(* PLC project Generated.project, CODESYS CODESYS V3.5 SP19 Patch 1 *)
(* stored: creationDateTime 2026-09-06T13:00:42.426166, modificationDateTime 2026-09-06T13:00:42.426166 *)

(* values of E_Mode: DISABLE: Mode Désactivé / Veille de sécurité (sorties bloquées); MAINT_N1: Manuel Niveau 1 : Pilotage unitaire avec toutes sécurités actives; MAINT_N2: Manuel Niveau 2 : Pilotage dégradé (droits étendus + bypasses autorisés); SEMI_AUTO: Mode Semi-Automatique (séquenceur automatique) *)

{attribute 'qualified_only'}
{attribute 'strict'}
TYPE E_Mode : (DISABLE := 0, MAINT_N1 := 1, MAINT_N2 := 2, SEMI_AUTO := 3);
END_TYPE

(* ======================================================================= 🧩 ST_Fault — Brique socle défaut (2 vues : live + latchée) ─────────────────────────────────────────────────────────────── 🎯 Rôle : porter l'état défaut d'un composant, applicable dans TOUS les cas (acquittable ou non), sans brique warning séparée. • Vue LIVE (Error / ErrorId) : suit la cause, retombe seule à 0. • Vue LATCHÉE (Latched / LatchedId): mémorisée au défaut, reste jusqu'au front Reset. Le choix acquittable / non-acquittable se fait PAR CAUSE (ST_FaultCause.Latching), jamais par bloc. 🔒 Sécurité : interlock TOUJOURS sur la cause brute (Error / ErrorId), jamais sur l'acquittement. Reset TOUJOURS effectif, jamais conditionné (std §9). 🧬 Composition : brique de base réutilisable — sortie de FB, struct métier, GVL. Texte IHM NON stocké ici : dérivé côté IHM depuis LatchedId / ErrorId. 📄 Doc : DOC/STDS/CODE_QUALITY_STANDARDS.md §2quinquies / §9 ======================================================================= *)
TYPE ST_Fault : STRUCT
  Error : BOOL;  (* <-- [DIAG] vue LIVE : au moins une cause présente maintenant *)
  ErrorId : WORD;  (* <-- [DIAG] bitfield des causes présentes maintenant (0 si aucune) *)
  Latched : BOOL;  (* <-- [DIAG] vue LATCHÉE : défaut non acquitté, reste jusqu'au front Reset *)
  LatchedId : WORD;  (* <-- [DIAG] ErrorId figé à l'apparition du défaut, effacé au Reset *)
END_STRUCT;
END_TYPE

(* ======================================================================= 🧩 ST_FaultCause — Cause élémentaire alimentant ST_Fault (socle FB_FaultCore) ─────────────────────────────────────────────────────────────── 🎯 Rôle : une cause exprimée EN CLAIR (BOOL + libellé), sans bitfield ni masque. Le FB métier remplit une liste (ARRAY[0..15] OF ST_FaultCause) ; le socle FB_FaultCore en déduit ST_Fault (vue live + vue latchée). 🔒 Sécurité : interlock TOUJOURS sur Active (cause brute), jamais sur le latch. Latching = TRUE → la cause ARME la vue latchée (défaut à acquitter). Latching = FALSE → la cause n'alimente que la vue live (retombe seule). Fail-safe : une cause laissée à Latching=FALSE reste visible en live — pour la rendre acquittable, il faut le déclarer explicitement. 📄 Doc : DOC/STDS/CODE_QUALITY_STANDARDS.md §2quinquies / §9 ======================================================================= *)
TYPE ST_FaultCause : STRUCT
  Active : BOOL;  (* 1 = cause présente maintenant (interlock sur cette valeur) *)
  Latching : BOOL;  (* 1 = cause à acquitter (arme Latched) ; 0 = live seulement *)
  Texte : STRING;  (* libellé prêt IHM (non stocké dans ST_Fault, dérivé côté IHM) *)
END_STRUCT;
END_TYPE

(* ======================================================================= ⚙️ ST_fbWinchLoadEstimator_SpeedCfg — Configuration des plages de vitesse linéaire ─────────────────────────────────────────────────────────────── 🎯 Rôle : Caractérisation des plages de vitesse mesurée par palier (m/s) 📄 Doc métier : DOC/AF/AF_Partie-10_Fonction_Winch_v2.1.md ======================================================================= *)
TYPE ST_fbWinchLoadEstimator_SpeedCfg : STRUCT
  MaxMeasuredSpeedMps : REAL;  (* Vitesse maximale mesuree de reference (m/s) *)
  SpeedBandMaxMps : ARRAY[1..5] OF REAL;  (* Plafonds vitesse mesuree par palier (m/s) *)
  SpeedBandHysteresisMps : REAL;  (* Hysteresis anti-battement classement vitesse (m/s) *)
END_STRUCT;
END_TYPE

(* ======================================================================= 📊 ST_fbWinchLoadEstimator_Table — Table empirique de charge estimée ─────────────────────────────────────────────────────────────── 🎯 Rôle : Matrice 5x5 d'estimation de charge (palier commandé x bande vitesse) 📄 Doc métier : DOC/AF/AF_Partie-10_Fonction_Winch_v2.1.md ======================================================================= *)
TYPE ST_fbWinchLoadEstimator_Table : STRUCT
  IsConfigured : BOOL;  (* Validation explicite de la table *)
  LoadPctByStepAndSpeedBand : ARRAY[1..5] OF ARRAY[1..5] OF REAL;  (* Matrice [palier][bande_vitesse] charge (%) *)
END_STRUCT;
END_TYPE

(* ======================================================================= 📊 FB_WinchLoadEstimator — Estimation empirique de charge treuil ─────────────────────────────────────────────────────────────── 🎯 Rôle : Estimation informative de la charge par croisement palier/vitesse 📄 Doc métier : DOC/AF/AF_Partie-10_Fonction_Winch_v2.1.md 🔌 Interface : Brique de diagnostic/mesure (1 instance par treuil) 🔒 Sécurité : Aucune commande moteur ni action sur SafeStop (information IHM) ======================================================================= *)
FUNCTION_BLOCK FB_WinchLoadEstimator
  VAR_INPUT
    Enable : BOOL;  (* === COMMANDES ET CONSIGNES === --> [CMD] Autorisation generale FB *)
    Reset : BOOL;  (* --> [CMD] Acquittement defaut sur front *)
    Mode : E_Mode;  (* --> [CMD] Mode d'exploitation actif *)
    ActiveSpeedStep : INT;  (* --> [CMD] Palier commande actif (0..5) *)
    PowerContactorEngaged : BOOL;  (* === SECOURS ET HARDWARE === --> [SAFE] Chaine AU rearmee et puissance OK *)
    MeasuredSpeedMps : REAL;  (* --> [HW] Vitesse cable absolue (m/s) *)
    MeasuredSpeedSignedMps : REAL;  (* --> [HW] Vitesse signee (+: montee, -: descente) (m/s) *)
    SpeedConfig : ST_fbWinchLoadEstimator_SpeedCfg;  (* === REGLAGES ET TABLES === --> [CFG] Configuration des plages de vitesse *)
    LoadTable : ST_fbWinchLoadEstimator_Table;  (* --> [CFG] Table empirique d'estimation 5x5 *)
  END_VAR
  VAR_OUTPUT
    Ready : BOOL;  (* === ETATS IEC ET SYNOPTIQUE === <-- [STAT] FB pret a fonctionner *)
    Fault : ST_Fault;  (* 🧩 Statut transverse (forme cible ST_Fault) *)
    SpeedBand : INT;  (* === DIAGNOSTICS ET ESTIMATIONS === <-- [DIAG] Bande de vitesse courante (0..5) *)
    EstimatedLoadPct : REAL;  (* <-- [DIAG] Estimation de charge (0..100%) *)
    Configured : BOOL;  (* <-- [STAT] Table explicitement validee *)
    Ascending : BOOL;  (* <-- [STAT] Ascending effective mesuree en cours *)
  END_VAR
  VAR
    ResetEdge : R_TRIG;  (* === DETECTEURS ET TIMERS INTERNES === . [LOC] Detecteur front montant Reset *)
    PreviousSpeedBand : INT;  (* === VARIABLES LOCALES CALCULÉES === . [LOC] Memoire bande de vitesse cycle precedent *)
    HasPreviousBand : BOOL;  (* . [LOC] Indicateur premiere bande memorisee *)
    SelectedLoadPct : REAL;  (* . [LOC] Valeur de charge extraite de la table *)
    ConfigOrSpeedFault : BOOL;  (* . [LOC] Latch défaut configuration / vitesse *)
    instFault : FB_FaultCore;  (* === SOCLE DEFAUT === * [INST] Socle défaut transverse *)
    instCauses : ARRAY[0..15] OF ST_FaultCause;  (* . [LOC] Table des causes nommées *)
  END_VAR

            

// === IMPLEMENTATION ===

{region "§1 Causes & Socle Défaut (évalué en continu)"}
// 🔑 1. FRONTS
ResetEdge(CLK := Reset);

IF ResetEdge.Q AND (MeasuredSpeedMps >= 0.0) THEN
    ConfigOrSpeedFault := FALSE;
END_IF;

instCauses[0].Active   := ConfigOrSpeedFault;
instCauses[0].Latching := TRUE;
instCauses[0].Texte    := 'Parametrage ou vitesse estimation charge invalide';

// Appel du socle de défaut
instFault(Enable := Enable, Reset := Reset, Causes := instCauses);
Fault := instFault.Fault;
{endregion}

{region "§2 Gate neutralisation"}
// 🛑 2. GATE
IF NOT Enable OR NOT PowerContactorEngaged THEN
    Ready := FALSE;
    SpeedBand := 0;
    EstimatedLoadPct := 0.0;
    Configured := FALSE;
    Ascending := FALSE;
    HasPreviousBand := FALSE;
    RETURN;
END_IF;

Ready := Enable AND NOT Fault.Latched;
Configured := LoadTable.IsConfigured;
Ascending := (MeasuredSpeedSignedMps > 0.0);
{endregion}

{region "§3 Classement vitesse"}
// 📏 3. CLASSEMENT DE LA VITESSE — hystérésis autour des 4 frontières.
IF (MeasuredSpeedMps < 0.0) OR (SpeedConfig.MaxMeasuredSpeedMps <= 0.0) THEN
    ConfigOrSpeedFault := TRUE;
    SpeedBand := 0;
ELSIF NOT HasPreviousBand THEN
    IF MeasuredSpeedMps <= SpeedConfig.SpeedBandMaxMps[1] THEN
        PreviousSpeedBand := 1;
    ELSIF MeasuredSpeedMps <= SpeedConfig.SpeedBandMaxMps[2] THEN
        PreviousSpeedBand := 2;
    ELSIF MeasuredSpeedMps <= SpeedConfig.SpeedBandMaxMps[3] THEN
        PreviousSpeedBand := 3;
    ELSIF MeasuredSpeedMps <= SpeedConfig.SpeedBandMaxMps[4] THEN
        PreviousSpeedBand := 4;
    ELSE
        PreviousSpeedBand := 5;
    END_IF;
    HasPreviousBand := TRUE;
    SpeedBand := PreviousSpeedBand;
ELSE
    IF PreviousSpeedBand < 1 OR PreviousSpeedBand > 5 THEN
        PreviousSpeedBand := 1;
        ConfigOrSpeedFault := TRUE;
    END_IF;

    IF PreviousSpeedBand < 5 THEN
        IF MeasuredSpeedMps > (SpeedConfig.SpeedBandMaxMps[PreviousSpeedBand]
                               + SpeedConfig.SpeedBandHysteresisMps) THEN
            PreviousSpeedBand := PreviousSpeedBand + 1;
        END_IF;
    END_IF;
    IF PreviousSpeedBand > 1 THEN
        IF MeasuredSpeedMps < (SpeedConfig.SpeedBandMaxMps[PreviousSpeedBand - 1]
                               - SpeedConfig.SpeedBandHysteresisMps) THEN
            PreviousSpeedBand := PreviousSpeedBand - 1;
        END_IF;
    END_IF;
    SpeedBand := PreviousSpeedBand;
END_IF;
{endregion}

{region "§4 Lecture table"}
// 📊 4. LECTURE TABLE
EstimatedLoadPct := 0.0;
IF Configured THEN
    IF Ascending THEN
        IF ActiveSpeedStep >= 1 THEN
            IF ActiveSpeedStep <= 5 THEN
                IF SpeedBand >= 1 THEN
                    IF SpeedBand <= 5 THEN
                        SelectedLoadPct := LoadTable.LoadPctByStepAndSpeedBand[ActiveSpeedStep][SpeedBand];
                        IF (SelectedLoadPct < 0.0) OR (SelectedLoadPct > 100.0) THEN
                            ConfigOrSpeedFault := TRUE;
                        ELSE
                            EstimatedLoadPct := SelectedLoadPct;
                        END_IF;
                    END_IF;
                END_IF;
            END_IF;
        END_IF;
    END_IF;
END_IF;
{endregion}

          
END_FUNCTION_BLOCK

(* ======================================================================= 🧩 FB_FaultCore — Socle de remplissage de ST_Fault (vue live + vue latchée) ─────────────────────────────────────────────────────────────── 🎯 Rôle : à partir d'une LISTE de causes en clair (ARRAY[0..15] OF ST_FaultCause), produire la brique ST_Fault : • Error / ErrorId : vue LIVE, suit les causes Active, retombe seule. • Latched / LatchedId: vue LATCHÉE, chaque bit figé à l'apparition d'une cause `Active AND Latching`, conservé jusqu'au front Reset. 🔒 Sécurité : - interlock TOUJOURS sur `Causes[i].Active` (cause brute), jamais sur le latch. - Reset TOUJOURS effectif, jamais conditionné (std §9) — agit même Enable=FALSE. - Latching=FALSE → cause visible en LIVE seulement (fail-safe : reste visible). - un défaut laté non acquitté reste publié même FB désactivé (pas d'effacement silencieux sur bascule Enable OFF→ON sans Reset). - une cause à acquitter réapparue re-arme son bit (ré-alarme). 🧬 Un seul socle, réutilisé par tout FB `standard` qui expose un ST_Fault. Pas de State, pas de Warning, pas de texte — hors périmètre de ce socle. 📄 Doc : DOC/STDS/CODE_QUALITY_STANDARDS.md §2quinquies / §9 ======================================================================= *)
FUNCTION_BLOCK FB_FaultCore
  VAR_INPUT
    Enable : BOOL;  (* --> [CMD] Autorisation générale du FB porteur *)
    Reset : BOOL;  (* --> [CMD] Front d'acquittement (jamais conditionné, §9) *)
    Causes : ARRAY[0..15] OF ST_FaultCause;  (* --> [CMD] Liste des causes en clair (Active / Latching / Texte) *)
  END_VAR
  VAR_OUTPUT
    Ready : BOOL;  (* <-- [STAT] FB porteur autorisé (= Enable) *)
    Fault : ST_Fault;  (* <-- [DIAG] Brique défaut (mappée 1:1 sur la sortie du FB porteur) *)
  END_VAR
  VAR
    ResetEdge : R_TRIG;  (* . [LOC] Front montant Reset *)
    Latch : ARRAY[0..15] OF BOOL;  (* . [LOC] Bit laté par cause, jusqu'au Reset *)
    i : INT;  (* . [LOC] Index de parcours de la liste *)
  END_VAR

            

{region "§1 Reset (front, toujours effectif)"}
// Front Reset : efface tous les latches. Jamais conditionné, agit même Enable=FALSE (§9).
Ready := Enable;
ResetEdge(CLK := Reset);
IF ResetEdge.Q THEN
    FOR i := 0 TO 15 DO Latch[i] := FALSE; END_FOR;
END_IF;
{endregion}

{region "§2 Vue LIVE — Error / ErrorId"}
// Bitfield des causes présentes MAINTENANT. Retombe seule à 0 quand les causes disparaissent.
// Non évaluée si Enable=FALSE (pas de lecture de cause hors autorisation).
Fault.ErrorId := 0;
IF Enable THEN
    FOR i := 0 TO 15 DO
        IF Causes[i].Active THEN
            Fault.ErrorId := Fault.ErrorId OR SHL(WORD#1, INT_TO_DWORD(i));
        END_IF;
    END_FOR;
END_IF;
Fault.Error := (Fault.ErrorId <> 0);
{endregion}

{region "§3 Armement des latches (causes à acquitter)"}
// Une cause Active ET Latching arme son bit ; le bit reste jusqu'au front Reset (§1),
// même si la cause disparaît. Réapparition => ré-armement (ré-alarme).
IF Enable THEN
    FOR i := 0 TO 15 DO
        IF Causes[i].Active AND Causes[i].Latching THEN
            Latch[i] := TRUE;
        END_IF;
    END_FOR;
END_IF;
{endregion}

{region "§4 Vue LATCHÉE — Latched / LatchedId"}
// Toujours publiée, y compris Enable=FALSE : un défaut non acquitté reste visible.
Fault.LatchedId := 0;
FOR i := 0 TO 15 DO
    IF Latch[i] THEN
        Fault.LatchedId := Fault.LatchedId OR SHL(WORD#1, INT_TO_DWORD(i));
    END_IF;
END_FOR;
Fault.Latched := (Fault.LatchedId <> 0);
{endregion}

          
END_FUNCTION_BLOCK
